(*
  This fb handles mechanical print unit corrections.
  - a 4p grid distortion
  - print unit bar banana correction
  NOTE: temperature extention of whole printbar is still handled in camera
*)
FUNCTION_BLOCK FB_FineAlignement EXTENDS FB_BasePrint
VAR
  // config
  _fPxResolution     : LREAL; // pixel resolution
  // corrections
  //-- 4 point PU deformation correction/distortion
  //    VISU setup point providing reference and correction (NOTE: persists settings internally)
  _fbPUCorrPoints    : ARRAY[1..4] OF FB_PointCorr;
  //-- banana correction
  _fT1 : LREAL;   // temperature 1
  _fT2 : LREAL;   // temperature 2
  _dx_middle : LREAL;  // correction in middle (for view only)
  _y_max : LREAL; // print unit width [mm]

  // helper
  lCtr     : UDINT;
  
  // unit test & debug
  _bUT_4p, _bUT_banana : BOOL;
  _sUTPoints_dx : ARRAY[0..nC_UT_cols, 0..nC_UT_rows] OF LREAL;
  _sUTPoints_dy : ARRAY[0..nC_UT_cols, 0..nC_UT_rows] OF LREAL;
END_VAR
VAR PERSISTENT
  //-- 4point correction
  _bEnable_4p : BOOL := TRUE;
  //  persistence of points see: FB_PointCorr
  //-- banana correction
  _bEnable_banana : BOOL := TRUE;
  _e_max_per_deltaT : LREAL := 0.01;  // [mm/°C]  TODO: use from config
END_VAR
VAR CONSTANT
  // Unit test configuration
  nC_UT_cols : DINT := 6;   // for test only
  nC_UT_rows : DINT := 5;   // for test only
END_VAR

// cyclic caluclation and view updates

//-- 4p correction
//    visu overrides (limitation rectancular point definition)
_fbPUCorrPoints[3].fX_Ref := _fbPUCorrPoints[1].fX_Ref;
_fbPUCorrPoints[4].fX_Ref := _fbPUCorrPoints[2].fX_Ref;
_fbPUCorrPoints[2].fY_Ref := _fbPUCorrPoints[1].fY_Ref;
_fbPUCorrPoints[4].fY_Ref := _fbPUCorrPoints[3].fY_Ref;
//    update view elements and handle inputs
FOR lCtr := 1 TO 4 DO
  _fbPUCorrPoints[lCtr](); 
END_FOR

//-- banana correction
// no cyclic update (here just for visu)
calc_banana_correction(x_pos:=0, y_pos:=_y_max/(2*1000), fT1:=_fT1, fT2:=_fT2, dx_corr=>_dx_middle);
_dx_middle := _dx_middle * 1000; // [m] --> [mm] for visu

// Unit test
IF _bUT_4p THEN _bUT_4p := FALSE; _test_4p(); END_IF
IF _bUT_banana THEN _bUT_banana := FALSE; _test_banana(); END_IF

METHOD PRIVATE _test_4p
VAR
  sPoint : ST_DeformationPoint;
  nCol, nRow : DINT;
  dx, dy : LREAL;       // correction in [m]
  dx_px, dy_px : DINT;  // correction in [px]
END_VAR
// generate internal grid
FOR nCol:=0 TO nC_UT_cols DO
  FOR nRow:=0 TO nC_UT_rows DO
    sPoint.col := nCol;
    sPoint.row := nRow;
    sPoint.x_ref := nCol * TO_DINT(GVL_Deformation.nC_GridPitch_X);
    sPoint.y_ref := nRow * TO_DINT(GVL_Deformation.nC_GridPitch_Y);
    sPoint.dx := 0;   // no previous deformation
    sPoint.dy := 0;   // no previous deformation
    // calc correction and apply to point
    calc_4p_correction(
        x_pos:=F_SubPixelToMeter(lPosSubPx:=sPoint.x_ref, fResSubPx:=_fPxResolution), 
        y_pos:=F_SubPixelToMeter(lPosSubPx:=sPoint.y_ref, fResSubPx:=_fPxResolution), 
        dx_corr=>dx, 
        dy_corr=>dy);
    dx_px := F_MeterToSubPixel(fPosMeter:=dx, fResoSubPx:=_fPxResolution);
    dy_px := F_MeterToSubPixel(fPosMeter:=dy, fResoSubPx:=_fPxResolution);
    // save corrected point
    _sUTPoints_dx[nCol, nRow] := dx_px;
    _sUTPoints_dy[nCol, nRow] := dy_px;
    // print corrected point
    LogInfo(
      F_Concat4(
        F_Concat4('[c/r] ', TO_STRING(sPoint.col), '/', TO_STRING(sPoint.row)),
        F_Concat6(' dx: ', TO_STRING(sPoint.dx), '>', TO_STRING(dx_px), ' [', TO_STRING(dx)),
        F_Concat6('  dy: ', TO_STRING(sPoint.dy), '>', TO_STRING(dy_px), ' [', TO_STRING(dy)),
        SEL(sPoint.dx<>dx_px OR sPoint.dy<>dy_px,'',' !!!')
      )
    );
  END_FOR  
END_FOR
END_METHOD

METHOD PRIVATE _test_banana
VAR
  sPoint : ST_DeformationPoint;
  nCol, nRow : DINT;
  dx, dy : LREAL;       // correction in [m]
  dx_px, dy_px : LREAL;  // correction in [px]
END_VAR
// generate internal grid
FOR nCol:=0 TO nC_UT_cols DO
  FOR nRow:=0 TO nC_UT_rows DO
    sPoint.col := nCol;
    sPoint.row := nRow;
    sPoint.x_ref := nCol * TO_DINT(GVL_Deformation.nC_GridPitch_X);
    sPoint.y_ref := nRow * TO_DINT(GVL_Deformation.nC_GridPitch_Y);
    sPoint.dx := 0;   // no previous deformation
    sPoint.dy := 0;   // no previous deformation
    
    // calc correction and apply to point
    calc_banana_correction(
        x_pos:=F_SubPixelToMeter(lPosSubPx:=sPoint.x_ref, fResSubPx:=_fPxResolution), 
        Y_pos:=F_SubPixelToMeter(lPosSubPx:=sPoint.y_ref, fResSubPx:=_fPxResolution),
        fT1 := 68,
        fT2 := 48, 
        dx_corr=>dx
    );
    dx_px := dx;
    dy_px := dy;
    // save corrected point (dx @y-pos)
    _sUTPoints_dx[nCol, nRow] := dx_px;
    _sUTPoints_dy[nCol, nRow] := F_SubPixelToMeter(lPosSubPx:=sPoint.y_ref, fResSubPx:=_fPxResolution)*1000;
    
    // print corrected point
    LogInfo(
      F_Concat4(
        F_Concat4('[c/r] ', TO_STRING(sPoint.col), '/', TO_STRING(sPoint.row)),
        F_Concat6(' dx: ', TO_STRING(sPoint.dx), '>', TO_STRING(TO_DINT(dx_px)), ' [', TO_STRING(dx)),
        F_Concat6('  dy: ', TO_STRING(sPoint.dy), '>', TO_STRING(TO_DINT(dy_px)), ' [', TO_STRING(dy)),
        SEL(sPoint.dx<>dx_px OR sPoint.dy<>dy_px,'',' !!!')
      )
    );
  END_FOR  
END_FOR
END_METHOD

(*
  Calculate grid point displacement for a distortion with 4 rectangular defined points.
  Uses 2-bilinear interpolation between the 4 rectancular reference points.
*)
METHOD PRIVATE calc_4p_correction : BOOL
VAR_INPUT
  x_pos   : LREAL;    // point x position [m]
  y_pos   : LREAL;    // point y position [m]
END_VAR
VAR_OUTPUT
  dx_corr : LREAL;    // point correction x [m]
  dy_corr : LREAL;    // point correction y [m]
END_VAR
VAR
  dx, dy : LREAL;     // difference between Calibration Points (rectangle)
  x1, x2, y1, y2 : LREAL;
  cx1, cx2, cy1, cy2 : LREAL;
  GPx, GPy : LREAL;
  CVx, CVy : LREAL;
  lErrCtr : UDINT;
END_VAR

// Grid point position
GPx := x_pos; 
GPy := y_pos;

// Interpolation in x
x1 := _fbPUCorrPoints[1].fX_Ref / 1000;    // [mm -> m]
x2 := _fbPUCorrPoints[2].fX_Ref / 1000;    // [mm -> m]
dx := x2-x1;
IF dx = 0 THEN F_Report_Error(ErrType:=EN_REPORT_ERROR_TYPE.Report_Error_0Pointer); RETURN; END_IF

cx1 := (x2-GPx)/dx * (_fbPUCorrPoints[1].fX / 1000) + (GPx-x1)/dx * (_fbPUCorrPoints[2].fX / 1000);
cx2 := (x2-GPx)/dx * (_fbPUCorrPoints[3].fX / 1000) + (GPx-x1)/dx * (_fbPUCorrPoints[4].fX / 1000);
cy1 := (x2-GPx)/dx * (_fbPUCorrPoints[1].fY / 1000) + (GPx-x1)/dx * (_fbPUCorrPoints[2].fY / 1000);
cy2 := (x2-GPx)/dx * (_fbPUCorrPoints[3].fY / 1000) + (GPx-x1)/dx * (_fbPUCorrPoints[4].fY / 1000);

// Interpolation in y
y1 := _fbPUCorrPoints[1].fY_Ref / 1000;    // [mm -> m]
y2 := _fbPUCorrPoints[3].fY_Ref / 1000;    // [mm -> m]
dy := y2-y1;
IF dy = 0 THEN F_Report_Error(ErrType:=EN_REPORT_ERROR_TYPE.Report_Error_0Pointer); RETURN; END_IF

// Calc interpolated 
CVx := (y2 - GPy)/dy * cx1 + (GPy-y1)/dy * cx2;
CVy := (y2 - GPy)/dy * cy1 + (GPy-y1)/dy * cy2;

// return accurate new correction only
dx_corr := CVx;
dy_corr := CVy;

calc_4p_correction := TRUE;
END_METHOD

(*
  Calculate grid point displacement for print unit banana deformation.
  2nd order approximation.
*)
METHOD PRIVATE calc_banana_correction : BOOL
VAR_INPUT
  x_pos   : LREAL;    // point x position [m]
  y_pos   : LREAL;    // point y position [m]
  fT1     : LREAL;    // temperature 1 [°C]
  fT2     : LREAL;    // temperature 2 [°C]
END_VAR
VAR_OUTPUT
  dx_corr : LREAL;    // point correction x [m]
END_VAR
VAR
  delta_T : LREAL;   // delta temperature
  e_max   : LREAL;   //
  a : LREAL;
  x_dash, y_dash : LREAL;
END_VAR
IF _y_max = 0 THEN RETURN; END_IF

x_dash := y_pos * 1000; // [m] -> [mm]

delta_T := fT2-fT1;
e_max   := delta_T * _e_max_per_deltaT;

a := 4 * e_max /  EXPT(_y_max, 2);
y_dash := a * EXPT(x_dash - (_y_max / 2), 2) - e_max;

// correction value
dx_corr := (y_dash / 1000);  // [mm] -> [m]

calc_banana_correction := TRUE;
END_METHOD

PROPERTY fT_PL1 : LREAL
SET
_fT1 := fT_PL1;
END_SET
END_PROPERTY

PROPERTY fT_PL2 : LREAL
SET
_fT2 := fT_PL2;
END_SET
END_PROPERTY

METHOD init : BOOL
VAR_INPUT
  fPxReso        : LREAL;   // pixel resolution
  fPuWidth       : LREAL;   // Print unit width [m]
END_VAR
_fPxResolution := fPxReso;
_y_max := fPuWidth * 1000;  // -> [mm]

// PU Deformation
_fbPUCorrPoints[1].init(aName:='P1', aUnit:='mm', fX_Min:=-5, fX_Max:=5, fY_Min:=-5, fY_Max:=5, fIncrStep:=0.1, 
                        bButnInvertX:=TRUE, bButnInvertY:=TRUE, bValInvertX:=TRUE, bValInvertY:=FALSE);
_fbPUCorrPoints[2].init(aName:='P2', aUnit:='mm', fX_Min:=-5, fX_Max:=5, fY_Min:=-5, fY_Max:=5, fIncrStep:=0.1,
                        bButnInvertX:=TRUE, bButnInvertY:=TRUE, bValInvertX:=TRUE, bValInvertY:=FALSE);
_fbPUCorrPoints[3].init(aName:='P3', aUnit:='mm', fX_Min:=-5, fX_Max:=5, fY_Min:=-5, fY_Max:=5, fIncrStep:=0.1,
                        bButnInvertX:=TRUE, bButnInvertY:=TRUE, bValInvertX:=TRUE, bValInvertY:=FALSE);
_fbPUCorrPoints[4].init(aName:='P4', aUnit:='mm', fX_Min:=-5, fX_Max:=5, fY_Min:=-5, fY_Max:=5, fIncrStep:=0.1,
                        bButnInvertX:=TRUE, bButnInvertY:=TRUE, bValInvertX:=TRUE, bValInvertY:=FALSE);
END_METHOD

(*
  Apply fine-alignement corrections to DefGrid point
*)
METHOD updateCorrection : BOOL
VAR_INPUT
  pPoint : POINTER TO ST_DeformationPointAccurate;
END_VAR
VAR
  x_pos, dx_corr, dx_tmp : LREAL; // [m]
  y_pos, dy_corr, dy_tmp : LREAL; // [m]
  lErrCtr : UDINT;
END_VAR
// grid point position
x_pos := F_SubPixelToMeter(lPosSubPx:=FC_LREAL_TO_DINT(pPoint^.x_ref, ADR(lErrCtr)), fResSubPx:=_fPxResolution);  // [px -> m] 
y_pos := F_SubPixelToMeter(lPosSubPx:=FC_LREAL_TO_DINT(pPoint^.y_ref, ADR(lErrCtr)), fResSubPx:=_fPxResolution);  // [px -> m]
dx_corr := 0;
dy_corr := 0;

// calc - 4 point sheet deformation (PU and machine mechanical distortions)
IF _bEnable_4p THEN
  calc_4p_correction(x_pos:=x_pos, y_pos:=y_pos, dx_corr=>dx_tmp, dy_corr=>dy_tmp);
  dx_corr := dx_tmp + dx_corr;
  dy_corr := dy_tmp + dy_corr;
END_IF

// calc - banana correction
IF _bEnable_banana THEN
  calc_banana_correction(x_pos:=x_pos, y_pos:=y_pos, fT1:=_fT1, fT2:=_fT2, dx_corr=>dx_tmp);
  dx_corr := dx_tmp + dx_corr;
END_IF
// apply new correction to deformation correction 
pPoint^.dx := pPoint^.dx + F_MeterToSubPixelReal(fPosMeter:=dx_corr, fResoSubPx:=_fPxResolution);
pPoint^.dy := pPoint^.dy + F_MeterToSubPixelReal(fPosMeter:=dy_corr, fResoSubPx:=_fPxResolution);

updateCorrection := TRUE;
END_METHOD

END_FUNCTION_BLOCK

(* stored: Version 1.1.0.1, ProductVersion 3.1.4024.3
   POU FB_FineAlignement: Id {b0fdbfcd-2a71-4ede-b938-0e28dbf7b80d}, SpecialFunc None
   Method _test_4p: Id {6f0fa0b6-cc58-4465-bff5-26ae640a97c0}
   Method _test_banana: Id {cdda5b50-a20e-4ef0-8e55-027af444ef1f}
   Method calc_4p_correction: Id {c5b8318f-9300-4b60-afbb-0f066a2ad2b7}
   Method calc_banana_correction: Id {cd11fc31-cdd1-4fff-a3a1-69aafb3db5bd}
   Property fT_PL1: Id {b286c81c-0aff-4511-94c9-d4cc9bd4439b}
   Set Set: Id {c98c4823-db0a-4cb5-8e5c-1cb8271580d0}
   Property fT_PL2: Id {54ff08d7-dae5-4a96-a73a-97aa019a8e38}
   Set Set: Id {1684f327-46b0-49b3-a6db-fbee77699606}
   Method init: Id {22d51a6a-e008-40d7-a511-92f228aee50f}
   Method updateCorrection: Id {67567b6c-ad9f-4c43-b042-ce1ae67d99c3} *)
